// TIA Portal V20 export
FUNCTION "FC_AnalogInputConfig" : Void   // FC35, SCL
{ S7_Optimized_Access := 'TRUE' }
// stored: SetENOAutomatically false
BEGIN
   REGION Description header 
       //==================================================================================
       // POSALUX Swiss SA / (C) Copyright 2025
       //----------------------------------------------------------------------------------
       // Title: FC_AnalogInputConfig
       // Comment/Function:
       //
       // Author: Fabien Waldt
       // Engineering: TIA Portal v17
       //----------------------------------------------------------------------------------
       // Change log table:
       // Version  | Date     | Expert in charge | Changes applied
       // ---------|----------|------------------|------------------------------------
       // 00.00.01 | 20250312 | WFA              | First released version
       // ==================================================================================
   END_REGION

   REGION Laser_Power_Meter
       "DB_AnalogInputDataPLC".Laser_Power_Meter.EnableAlarmMin   := FALSE;
       "DB_AnalogInputDataPLC".Laser_Power_Meter.EnableWarningMin := FALSE;
       "DB_AnalogInputDataPLC".Laser_Power_Meter.EnableWarningMax := FALSE;
       "DB_AnalogInputDataPLC".Laser_Power_Meter.EnableAlarmMax   := FALSE;
   END_REGION

   REGION Axis_B_Clamping_Part
       "DB_AnalogInputDataPLC".Axis_B_Clamping_Part.EnableAlarmMin   := FALSE;
       "DB_AnalogInputDataPLC".Axis_B_Clamping_Part.EnableWarningMin := FALSE;
       "DB_AnalogInputDataPLC".Axis_B_Clamping_Part.EnableWarningMax := FALSE;
       "DB_AnalogInputDataPLC".Axis_B_Clamping_Part.EnableAlarmMax   := FALSE;
   END_REGION

   REGION Laser_Air_Pressure_Process
       "DB_AnalogInputDataPLC".Laser_Air_Pressure_Process.EnableAlarmMin   := TRUE;
       "DB_AnalogInputDataPLC".Laser_Air_Pressure_Process.EnableWarningMin := TRUE;
       "DB_AnalogInputDataPLC".Laser_Air_Pressure_Process.EnableWarningMax := TRUE;
       "DB_AnalogInputDataPLC".Laser_Air_Pressure_Process.EnableAlarmMax   := TRUE;
   END_REGION

   REGION Inlet_Air_Pressure
       "DB_AnalogInputDataPLC".Inlet_Air_Pressure.EnableAlarmMin   := TRUE;
       "DB_AnalogInputDataPLC".Inlet_Air_Pressure.EnableWarningMin := TRUE;
       "DB_AnalogInputDataPLC".Inlet_Air_Pressure.EnableWarningMax := TRUE;
       "DB_AnalogInputDataPLC".Inlet_Air_Pressure.EnableAlarmMax   := TRUE;
   END_REGION

   REGION Ambiant_Temperature
       "DB_AnalogInputDataPLC".Ambiant_Temperature.EnableAlarmMin   := TRUE;
       "DB_AnalogInputDataPLC".Ambiant_Temperature.EnableWarningMin := TRUE;
       "DB_AnalogInputDataPLC".Ambiant_Temperature.EnableWarningMax := TRUE;
       "DB_AnalogInputDataPLC".Ambiant_Temperature.EnableAlarmMax   := TRUE;
   END_REGION

   REGION Machine_Temperature
       "DB_AnalogInputDataPLC".Machine_Temperature.EnableAlarmMin   := TRUE;
       "DB_AnalogInputDataPLC".Machine_Temperature.EnableWarningMin := TRUE;
       "DB_AnalogInputDataPLC".Machine_Temperature.EnableWarningMax := TRUE;
       "DB_AnalogInputDataPLC".Machine_Temperature.EnableAlarmMax   := TRUE;
   END_REGION

   REGION Cold_Water_Temperature_Input
       "DB_AnalogInputDataPLC".Cold_Water_Temperature_Input.EnableAlarmMin   := TRUE;
       "DB_AnalogInputDataPLC".Cold_Water_Temperature_Input.EnableWarningMin := TRUE;
       "DB_AnalogInputDataPLC".Cold_Water_Temperature_Input.EnableWarningMax := TRUE;
       "DB_AnalogInputDataPLC".Cold_Water_Temperature_Input.EnableAlarmMax   := TRUE;
   END_REGION

   REGION Cold_Water_Temperature_Output
       "DB_AnalogInputDataPLC".Cold_Water_Temperature_Output.EnableAlarmMin   := TRUE;
       "DB_AnalogInputDataPLC".Cold_Water_Temperature_Output.EnableWarningMin := TRUE;
       "DB_AnalogInputDataPLC".Cold_Water_Temperature_Output.EnableWarningMax := TRUE;
       "DB_AnalogInputDataPLC".Cold_Water_Temperature_Output.EnableAlarmMax   := TRUE;
   END_REGION

   REGION X_Axis_Temperature_PT1000
       "DB_AnalogInputDataPLC".X_Axis_Temperature_PT1000.EnableAlarmMin   := FALSE; //WFA
       "DB_AnalogInputDataPLC".X_Axis_Temperature_PT1000.EnableWarningMin := FALSE; //WFA
       "DB_AnalogInputDataPLC".X_Axis_Temperature_PT1000.EnableWarningMax := TRUE;
       "DB_AnalogInputDataPLC".X_Axis_Temperature_PT1000.EnableAlarmMax   := TRUE;
   END_REGION

   REGION Y_Axis_Temperature_PT1000
       "DB_AnalogInputDataPLC".Y_Axis_Temperature_PT1000.EnableAlarmMin   := FALSE; //WFA
       "DB_AnalogInputDataPLC".Y_Axis_Temperature_PT1000.EnableWarningMin := FALSE; //WFA
       "DB_AnalogInputDataPLC".Y_Axis_Temperature_PT1000.EnableWarningMax := TRUE;
       "DB_AnalogInputDataPLC".Y_Axis_Temperature_PT1000.EnableAlarmMax   := TRUE;
   END_REGION
   REGION X_Axis_Temperature_PTC
       "DB_AnalogInputDataPLC".X_Axis_Temperature_PTC.EnableAlarmMin   := FALSE;
       "DB_AnalogInputDataPLC".X_Axis_Temperature_PTC.EnableWarningMin := FALSE;
       "DB_AnalogInputDataPLC".X_Axis_Temperature_PTC.EnableWarningMax := FALSE;
       "DB_AnalogInputDataPLC".X_Axis_Temperature_PTC.EnableAlarmMax   := FALSE;
   END_REGION

   REGION Y_Axis_Temperature_PTC
       "DB_AnalogInputDataPLC".Y_Axis_Temperature_PTC.EnableAlarmMin   := FALSE;
       "DB_AnalogInputDataPLC".Y_Axis_Temperature_PTC.EnableWarningMin := FALSE;
       "DB_AnalogInputDataPLC".Y_Axis_Temperature_PTC.EnableWarningMax := FALSE;
       "DB_AnalogInputDataPLC".Y_Axis_Temperature_PTC.EnableAlarmMax   := FALSE;
   END_REGION

   REGION Nozzle_Overpressure
       "DB_AnalogInputDataPLC".Nozzle_Overpressure.EnableAlarmMin   := TRUE;
       "DB_AnalogInputDataPLC".Nozzle_Overpressure.EnableWarningMin := TRUE;
       "DB_AnalogInputDataPLC".Nozzle_Overpressure.EnableWarningMax := TRUE;
       "DB_AnalogInputDataPLC".Nozzle_Overpressure.EnableAlarmMax   := TRUE;
   END_REGION

   REGION Optical_Path_Overpressure
       "DB_AnalogInputDataPLC".Optical_Path_Overpressure.EnableAlarmMin   := TRUE;
       "DB_AnalogInputDataPLC".Optical_Path_Overpressure.EnableWarningMin := TRUE;
       "DB_AnalogInputDataPLC".Optical_Path_Overpressure.EnableWarningMax := TRUE;
       "DB_AnalogInputDataPLC".Optical_Path_Overpressure.EnableAlarmMax   := TRUE;
   END_REGION

   REGION Laser_Head_Overpressure
       "DB_AnalogInputDataPLC".Laser_Head_Overpressure.EnableAlarmMin   := TRUE;
       "DB_AnalogInputDataPLC".Laser_Head_Overpressure.EnableWarningMin := TRUE;
       "DB_AnalogInputDataPLC".Laser_Head_Overpressure.EnableWarningMax := TRUE;
       "DB_AnalogInputDataPLC".Laser_Head_Overpressure.EnableAlarmMax   := TRUE;
   END_REGION

   REGION ZL_Axis_Overpressure
       "DB_AnalogInputDataPLC".ZL_Axis_Overpressure.EnableAlarmMin   := TRUE;
       "DB_AnalogInputDataPLC".ZL_Axis_Overpressure.EnableWarningMin := TRUE;
       "DB_AnalogInputDataPLC".ZL_Axis_Overpressure.EnableWarningMax := TRUE;
       "DB_AnalogInputDataPLC".ZL_Axis_Overpressure.EnableAlarmMax   := TRUE;
   END_REGION

   REGION XY_Axis_Overpressure
       "DB_AnalogInputDataPLC".XY_Axis_Overpressure.EnableAlarmMin   := TRUE;
       "DB_AnalogInputDataPLC".XY_Axis_Overpressure.EnableWarningMin := TRUE;
       "DB_AnalogInputDataPLC".XY_Axis_Overpressure.EnableWarningMax := TRUE;
       "DB_AnalogInputDataPLC".XY_Axis_Overpressure.EnableAlarmMax   := TRUE;
   END_REGION

   REGION Left_Aspiration
       "DB_AnalogInputDataPLC".Left_Aspiration.EnableAlarmMin   := TRUE;
       "DB_AnalogInputDataPLC".Left_Aspiration.EnableWarningMin := TRUE;
       "DB_AnalogInputDataPLC".Left_Aspiration.EnableWarningMax := TRUE;
       "DB_AnalogInputDataPLC".Left_Aspiration.EnableAlarmMax   := TRUE;
   END_REGION

   REGION Right_Aspiration
       "DB_AnalogInputDataPLC".Right_Aspiration.EnableAlarmMin   := TRUE;
       "DB_AnalogInputDataPLC".Right_Aspiration.EnableWarningMin := TRUE;
       "DB_AnalogInputDataPLC".Right_Aspiration.EnableWarningMax := TRUE;
       "DB_AnalogInputDataPLC".Right_Aspiration.EnableAlarmMax   := TRUE;
   END_REGION

   REGION Clim_Temperature
       "DB_AnalogInputDataPLC".Clim_Temperature.EnableAlarmMin   := FALSE;
       "DB_AnalogInputDataPLC".Clim_Temperature.EnableWarningMin := FALSE;
       "DB_AnalogInputDataPLC".Clim_Temperature.EnableWarningMax := FALSE;
       "DB_AnalogInputDataPLC".Clim_Temperature.EnableAlarmMax   := FALSE;
   END_REGION

   REGION Sensor_Controller_Station1
       "DB_AnalogInputDataPLC".Sensor_Controller_Station1.EnableAlarmMin   := FALSE;
       "DB_AnalogInputDataPLC".Sensor_Controller_Station1.EnableWarningMin := FALSE;
       "DB_AnalogInputDataPLC".Sensor_Controller_Station1.EnableWarningMax := FALSE;
       "DB_AnalogInputDataPLC".Sensor_Controller_Station1.EnableAlarmMax   := FALSE;
   END_REGION

   REGION Cabinet_Temperature
       "DB_AnalogInputDataPLC".Cabinet_Temperature.EnableAlarmMin   := FALSE;
       "DB_AnalogInputDataPLC".Cabinet_Temperature.EnableWarningMin := FALSE;
       "DB_AnalogInputDataPLC".Cabinet_Temperature.EnableWarningMax := FALSE;
       "DB_AnalogInputDataPLC".Cabinet_Temperature.EnableAlarmMax   := FALSE;
   END_REGION
END_FUNCTION
